FUNCTION INTERNAL Mc2DirectionConvertTo : Tc2_Mc2.Mc_Direction
VAR_INPUT
	direction : MotionDirection;
END_VAR

CASE direction OF
	MotionDirection.Positive: Mc2DirectionConvertTo := Tc2_Mc2.Mc_Direction.Mc_Positive_Direction;
	MotionDirection.ShortestWay: Mc2DirectionConvertTo := Tc2_Mc2.Mc_Direction.Mc_Shortest_Way;
	MotionDirection.Negative: Mc2DirectionConvertTo := Tc2_Mc2.Mc_Direction.Mc_Negative_Direction;
	MotionDirection.Current: Mc2DirectionConvertTo := Tc2_Mc2.Mc_Direction.Mc_Current_Direction;
	MotionDirection.Undefined: Mc2DirectionConvertTo := Tc2_Mc2.Mc_Direction.Mc_Undefined_Direction;
END_CASE

END_FUNCTION

(* stored: Version 1.1.0.1, ProductVersion 3.1.4026.13
   POU Mc2DirectionConvertTo: Id {db39b066-873b-4796-b598-e821da01cd37}, SpecialFunc None *)
